FUNCTION ArrayBool_TO_Byte : BYTE
VAR_INPUT
	In:				POINTER TO	BOOL;
	InLen:			INT;// sizeof(In)
END_VAR
VAR
END_VAR

IF InLen<>8 THEN
	RETURN;
END_IF

ArrayBool_TO_Byte.0:=In[0];
ArrayBool_TO_Byte.1:=In[1];
ArrayBool_TO_Byte.2:=In[2];
ArrayBool_TO_Byte.3:=In[3];
ArrayBool_TO_Byte.4:=In[4];
ArrayBool_TO_Byte.5:=In[5];
ArrayBool_TO_Byte.6:=In[6];
ArrayBool_TO_Byte.7:=In[7];

END_FUNCTION

(* stored: Version 1.1.0.1, ProductVersion 3.1.4024.3
   POU ArrayBool_TO_Byte: Id {c150da52-2745-4d62-9caa-e584d5ca1659}, SpecialFunc None *)
